PROGRAM MAIN
VAR
END_VAR

P_DMX_Master();
P_DMX_Slave();

END_PROGRAM

(* stored: Version 1.1.0.1, ProductVersion 3.1.4024.0
   POU MAIN: Id {453a2ca2-9df1-478f-bb2c-7d0d72d32f7c}, SpecialFunc None *)
